// TIA Portal V18 export
FUNCTION_BLOCK "Main_Safety_RTG1"   // FB1, F_LAD
{ S7_Optimized_Access := 'TRUE' }
VERSION : 0.1
// stored: AutoNumber false, IsIECCheckEnabled false, UDAEnableTagReadback false
   VAR
      ACK_GL_Instance : ACK_GL;
      FS_Room1_Instance : "FS_Room1";
      FS_Room2_Instance : "FS_Room2";
      FS_ACC_Instance : "FS_ACC";
      FS_VerticalBeam_Instance : "FS_VerticalBeam";
   END_VAR
BEGIN

REGION Network 1: 全局确认钝化
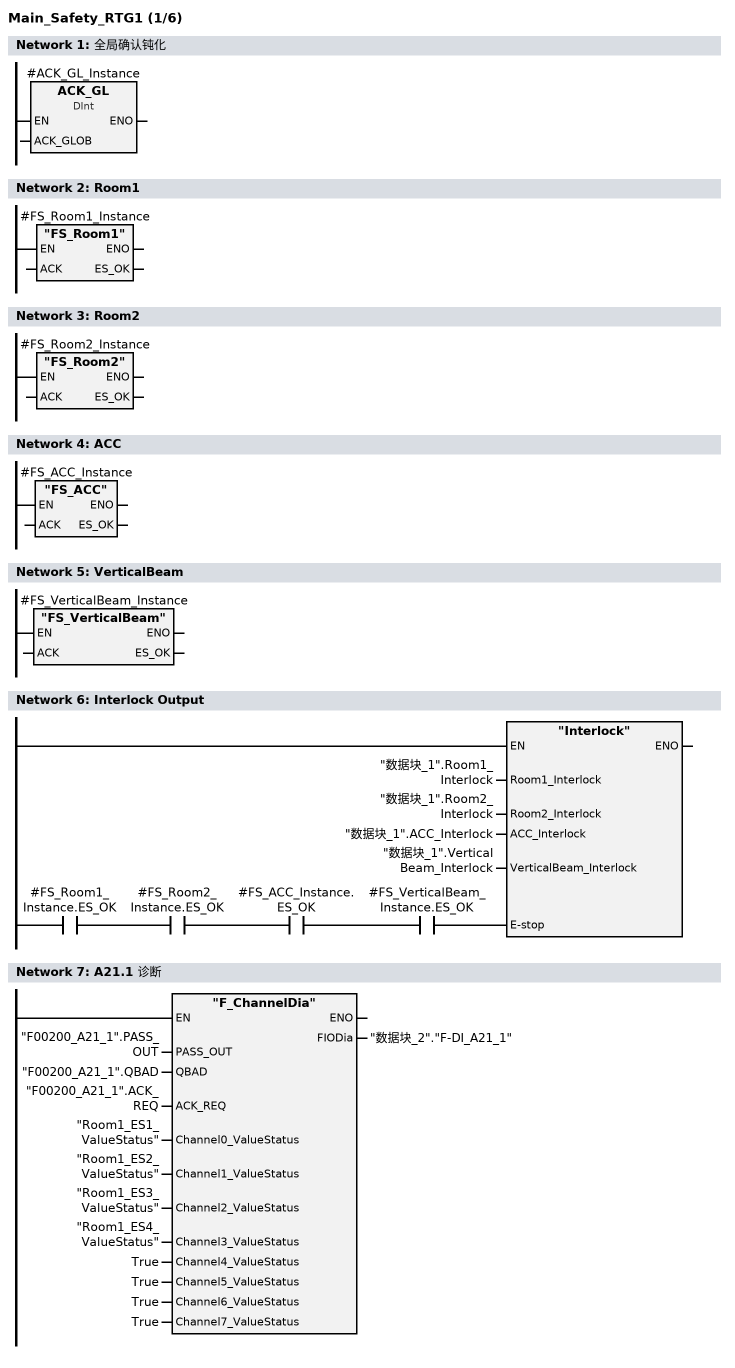
   RUNG wire#powerrail
      { S7_Templates := "codedbool_type := DInt" } #ACK_GL_Instance.ACK_GL(ACK_GLOB :=)
   END_RUNG
   // the same network as SCL:
   #ACK_GL_Instance();   // ACK_GL
END_REGION

REGION Network 2: Room1
   RUNG wire#powerrail
      #FS_Room1_Instance(ACK :=, ES_OK =>)
   END_RUNG
   // the same network as SCL:
   #FS_Room1_Instance();   // "FS_Room1"
END_REGION

REGION Network 3: Room2
   RUNG wire#powerrail
      #FS_Room2_Instance(ACK :=, ES_OK =>)
   END_RUNG
   // the same network as SCL:
   #FS_Room2_Instance();   // "FS_Room2"
END_REGION

REGION Network 4: ACC
   RUNG wire#powerrail
      #FS_ACC_Instance(ACK :=, ES_OK =>)
   END_RUNG
   // the same network as SCL:
   #FS_ACC_Instance();   // "FS_ACC"
END_REGION

REGION Network 5: VerticalBeam
   RUNG wire#powerrail
      #FS_VerticalBeam_Instance(ACK :=, ES_OK =>)
   END_RUNG
   // the same network as SCL:
   #FS_VerticalBeam_Instance();   // "FS_VerticalBeam"
END_REGION

REGION Network 6: Interlock Output
   RUNG wire#powerrail
      "Interlock"(Room1_Interlock := "数据块_1".Room1_Interlock, Room2_Interlock := "数据块_1".Room2_Interlock, ACC_Interlock := "数据块_1".ACC_Interlock, VerticalBeam_Interlock := "数据块_1".VerticalBeam_Interlock, "E-stop" := wire#w1)
   END_RUNG
   RUNG wire#powerrail
      Contact( #FS_Room1_Instance.ES_OK )
      Contact( #FS_Room2_Instance.ES_OK )
      Contact( #FS_ACC_Instance.ES_OK )
      Contact( #FS_VerticalBeam_Instance.ES_OK )
   END_RUNG wire#w1
   // the same network as SCL:
   "Interlock"(Room1_Interlock := "数据块_1".Room1_Interlock,
               Room2_Interlock := "数据块_1".Room2_Interlock,
               ACC_Interlock := "数据块_1".ACC_Interlock,
               VerticalBeam_Interlock := "数据块_1".VerticalBeam_Interlock,
               "E-stop" := #FS_Room1_Instance.ES_OK AND #FS_Room2_Instance.ES_OK AND #FS_ACC_Instance.ES_OK AND #FS_VerticalBeam_Instance.ES_OK);
END_REGION

REGION Network 7: A21.1 诊断
   RUNG wire#powerrail
      "F_ChannelDia"(PASS_OUT := "F00200_A21_1".PASS_OUT, QBAD := "F00200_A21_1".QBAD, ACK_REQ := "F00200_A21_1".ACK_REQ, Channel0_ValueStatus := "Room1_ES1_ValueStatus", Channel1_ValueStatus := "Room1_ES2_ValueStatus", Channel2_ValueStatus := "Room1_ES3_ValueStatus", Channel3_ValueStatus := "Room1_ES4_ValueStatus", Channel4_ValueStatus := True, Channel5_ValueStatus := True, Channel6_ValueStatus := True, Channel7_ValueStatus := True, FIODia => "数据块_2"."F-DI_A21_1")
   END_RUNG
   // the same network as SCL:
   "F_ChannelDia"(PASS_OUT := "F00200_A21_1".PASS_OUT,
                  QBAD := "F00200_A21_1".QBAD,
                  ACK_REQ := "F00200_A21_1".ACK_REQ,
                  Channel0_ValueStatus := "Room1_ES1_ValueStatus",
                  Channel1_ValueStatus := "Room1_ES2_ValueStatus",
                  Channel2_ValueStatus := "Room1_ES3_ValueStatus",
                  Channel3_ValueStatus := "Room1_ES4_ValueStatus",
                  Channel4_ValueStatus := True,
                  Channel5_ValueStatus := True,
                  Channel6_ValueStatus := True,
                  Channel7_ValueStatus := True,
                  FIODia => "数据块_2"."F-DI_A21_1");
END_REGION

REGION Network 8: A21.2 诊断
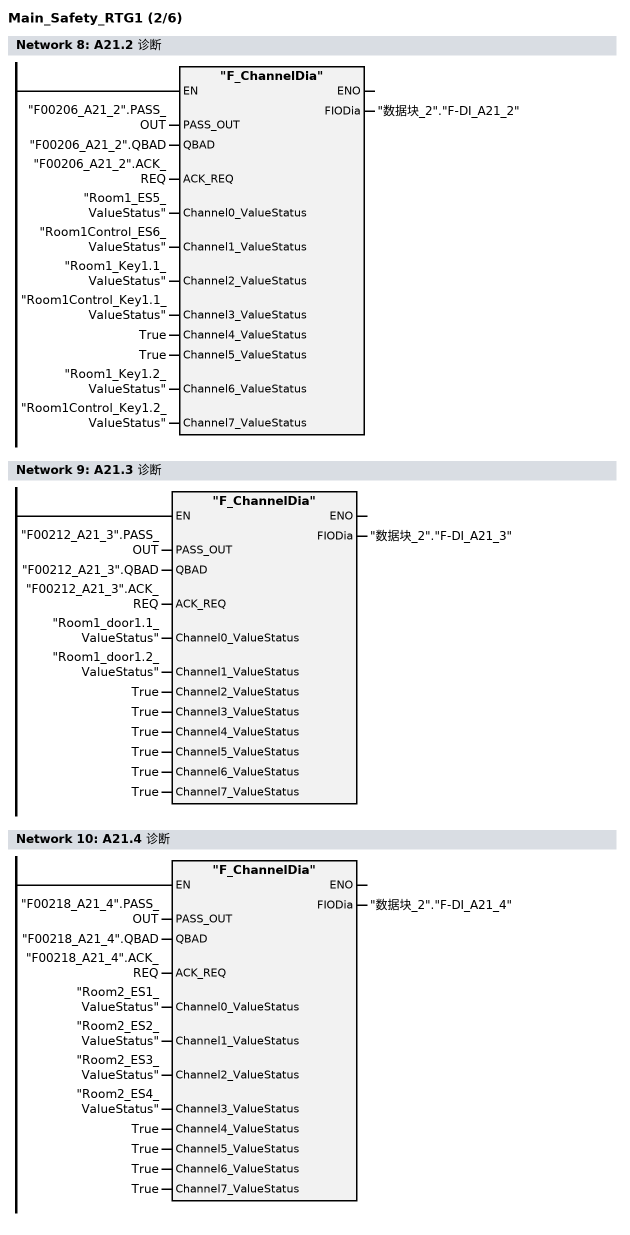
   RUNG wire#powerrail
      "F_ChannelDia"(PASS_OUT := "F00206_A21_2".PASS_OUT, QBAD := "F00206_A21_2".QBAD, ACK_REQ := "F00206_A21_2".ACK_REQ, Channel0_ValueStatus := "Room1_ES5_ValueStatus", Channel1_ValueStatus := "Room1Control_ES6_ValueStatus", Channel2_ValueStatus := "Room1_Key1.1_ValueStatus", Channel3_ValueStatus := "Room1Control_Key1.1_ValueStatus", Channel4_ValueStatus := True, Channel5_ValueStatus := True, Channel6_ValueStatus := "Room1_Key1.2_ValueStatus", Channel7_ValueStatus := "Room1Control_Key1.2_ValueStatus", FIODia => "数据块_2"."F-DI_A21_2")
   END_RUNG
   // the same network as SCL:
   "F_ChannelDia"(PASS_OUT := "F00206_A21_2".PASS_OUT,
                  QBAD := "F00206_A21_2".QBAD,
                  ACK_REQ := "F00206_A21_2".ACK_REQ,
                  Channel0_ValueStatus := "Room1_ES5_ValueStatus",
                  Channel1_ValueStatus := "Room1Control_ES6_ValueStatus",
                  Channel2_ValueStatus := "Room1_Key1.1_ValueStatus",
                  Channel3_ValueStatus := "Room1Control_Key1.1_ValueStatus",
                  Channel4_ValueStatus := True,
                  Channel5_ValueStatus := True,
                  Channel6_ValueStatus := "Room1_Key1.2_ValueStatus",
                  Channel7_ValueStatus := "Room1Control_Key1.2_ValueStatus",
                  FIODia => "数据块_2"."F-DI_A21_2");
END_REGION

REGION Network 9: A21.3 诊断
   RUNG wire#powerrail
      "F_ChannelDia"(PASS_OUT := "F00212_A21_3".PASS_OUT, QBAD := "F00212_A21_3".QBAD, ACK_REQ := "F00212_A21_3".ACK_REQ, Channel0_ValueStatus := "Room1_door1.1_ValueStatus", Channel1_ValueStatus := "Room1_door1.2_ValueStatus", Channel2_ValueStatus := True, Channel3_ValueStatus := True, Channel4_ValueStatus := True, Channel5_ValueStatus := True, Channel6_ValueStatus := True, Channel7_ValueStatus := True, FIODia => "数据块_2"."F-DI_A21_3")
   END_RUNG
   // the same network as SCL:
   "F_ChannelDia"(PASS_OUT := "F00212_A21_3".PASS_OUT,
                  QBAD := "F00212_A21_3".QBAD,
                  ACK_REQ := "F00212_A21_3".ACK_REQ,
                  Channel0_ValueStatus := "Room1_door1.1_ValueStatus",
                  Channel1_ValueStatus := "Room1_door1.2_ValueStatus",
                  Channel2_ValueStatus := True,
                  Channel3_ValueStatus := True,
                  Channel4_ValueStatus := True,
                  Channel5_ValueStatus := True,
                  Channel6_ValueStatus := True,
                  Channel7_ValueStatus := True,
                  FIODia => "数据块_2"."F-DI_A21_3");
END_REGION

REGION Network 10: A21.4 诊断
   RUNG wire#powerrail
      "F_ChannelDia"(PASS_OUT := "F00218_A21_4".PASS_OUT, QBAD := "F00218_A21_4".QBAD, ACK_REQ := "F00218_A21_4".ACK_REQ, Channel0_ValueStatus := "Room2_ES1_ValueStatus", Channel1_ValueStatus := "Room2_ES2_ValueStatus", Channel2_ValueStatus := "Room2_ES3_ValueStatus", Channel3_ValueStatus := "Room2_ES4_ValueStatus", Channel4_ValueStatus := True, Channel5_ValueStatus := True, Channel6_ValueStatus := True, Channel7_ValueStatus := True, FIODia => "数据块_2"."F-DI_A21_4")
   END_RUNG
   // the same network as SCL:
   "F_ChannelDia"(PASS_OUT := "F00218_A21_4".PASS_OUT,
                  QBAD := "F00218_A21_4".QBAD,
                  ACK_REQ := "F00218_A21_4".ACK_REQ,
                  Channel0_ValueStatus := "Room2_ES1_ValueStatus",
                  Channel1_ValueStatus := "Room2_ES2_ValueStatus",
                  Channel2_ValueStatus := "Room2_ES3_ValueStatus",
                  Channel3_ValueStatus := "Room2_ES4_ValueStatus",
                  Channel4_ValueStatus := True,
                  Channel5_ValueStatus := True,
                  Channel6_ValueStatus := True,
                  Channel7_ValueStatus := True,
                  FIODia => "数据块_2"."F-DI_A21_4");
END_REGION

REGION Network 11: A21.5 诊断
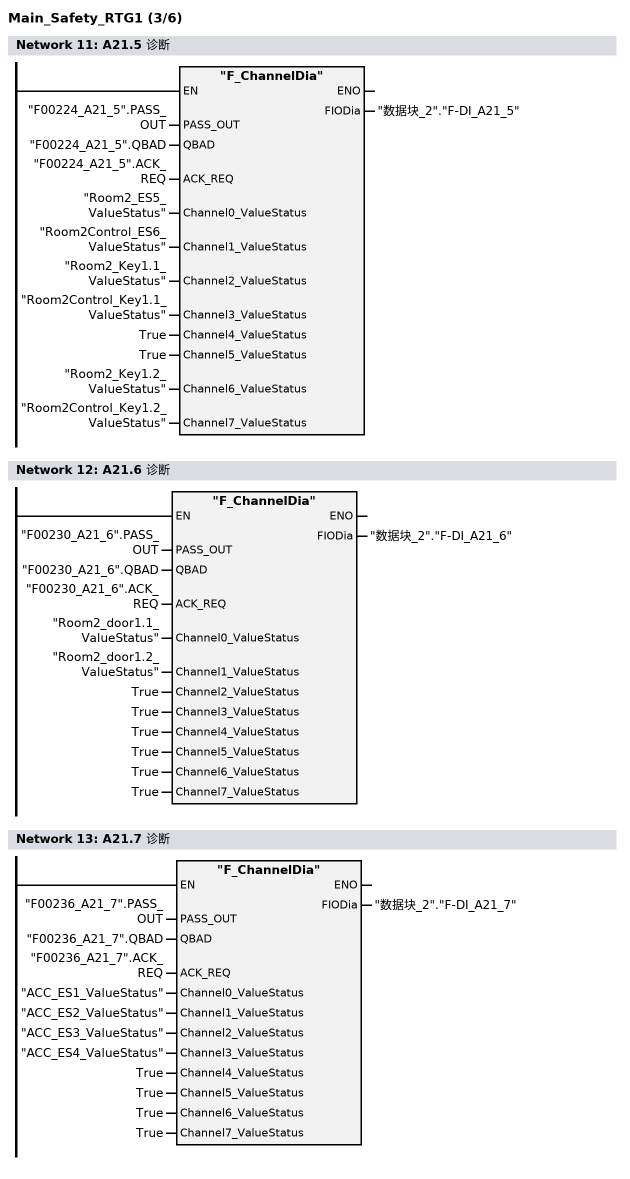
   RUNG wire#powerrail
      "F_ChannelDia"(PASS_OUT := "F00224_A21_5".PASS_OUT, QBAD := "F00224_A21_5".QBAD, ACK_REQ := "F00224_A21_5".ACK_REQ, Channel0_ValueStatus := "Room2_ES5_ValueStatus", Channel1_ValueStatus := "Room2Control_ES6_ValueStatus", Channel2_ValueStatus := "Room2_Key1.1_ValueStatus", Channel3_ValueStatus := "Room2Control_Key1.1_ValueStatus", Channel4_ValueStatus := True, Channel5_ValueStatus := True, Channel6_ValueStatus := "Room2_Key1.2_ValueStatus", Channel7_ValueStatus := "Room2Control_Key1.2_ValueStatus", FIODia => "数据块_2"."F-DI_A21_5")
   END_RUNG
   // the same network as SCL:
   "F_ChannelDia"(PASS_OUT := "F00224_A21_5".PASS_OUT,
                  QBAD := "F00224_A21_5".QBAD,
                  ACK_REQ := "F00224_A21_5".ACK_REQ,
                  Channel0_ValueStatus := "Room2_ES5_ValueStatus",
                  Channel1_ValueStatus := "Room2Control_ES6_ValueStatus",
                  Channel2_ValueStatus := "Room2_Key1.1_ValueStatus",
                  Channel3_ValueStatus := "Room2Control_Key1.1_ValueStatus",
                  Channel4_ValueStatus := True,
                  Channel5_ValueStatus := True,
                  Channel6_ValueStatus := "Room2_Key1.2_ValueStatus",
                  Channel7_ValueStatus := "Room2Control_Key1.2_ValueStatus",
                  FIODia => "数据块_2"."F-DI_A21_5");
END_REGION

REGION Network 12: A21.6 诊断
   RUNG wire#powerrail
      "F_ChannelDia"(PASS_OUT := "F00230_A21_6".PASS_OUT, QBAD := "F00230_A21_6".QBAD, ACK_REQ := "F00230_A21_6".ACK_REQ, Channel0_ValueStatus := "Room2_door1.1_ValueStatus", Channel1_ValueStatus := "Room2_door1.2_ValueStatus", Channel2_ValueStatus := True, Channel3_ValueStatus := True, Channel4_ValueStatus := True, Channel5_ValueStatus := True, Channel6_ValueStatus := True, Channel7_ValueStatus := True, FIODia => "数据块_2"."F-DI_A21_6")
   END_RUNG
   // the same network as SCL:
   "F_ChannelDia"(PASS_OUT := "F00230_A21_6".PASS_OUT,
                  QBAD := "F00230_A21_6".QBAD,
                  ACK_REQ := "F00230_A21_6".ACK_REQ,
                  Channel0_ValueStatus := "Room2_door1.1_ValueStatus",
                  Channel1_ValueStatus := "Room2_door1.2_ValueStatus",
                  Channel2_ValueStatus := True,
                  Channel3_ValueStatus := True,
                  Channel4_ValueStatus := True,
                  Channel5_ValueStatus := True,
                  Channel6_ValueStatus := True,
                  Channel7_ValueStatus := True,
                  FIODia => "数据块_2"."F-DI_A21_6");
END_REGION

REGION Network 13: A21.7 诊断
   RUNG wire#powerrail
      "F_ChannelDia"(PASS_OUT := "F00236_A21_7".PASS_OUT, QBAD := "F00236_A21_7".QBAD, ACK_REQ := "F00236_A21_7".ACK_REQ, Channel0_ValueStatus := "ACC_ES1_ValueStatus", Channel1_ValueStatus := "ACC_ES2_ValueStatus", Channel2_ValueStatus := "ACC_ES3_ValueStatus", Channel3_ValueStatus := "ACC_ES4_ValueStatus", Channel4_ValueStatus := True, Channel5_ValueStatus := True, Channel6_ValueStatus := True, Channel7_ValueStatus := True, FIODia => "数据块_2"."F-DI_A21_7")
   END_RUNG
   // the same network as SCL:
   "F_ChannelDia"(PASS_OUT := "F00236_A21_7".PASS_OUT,
                  QBAD := "F00236_A21_7".QBAD,
                  ACK_REQ := "F00236_A21_7".ACK_REQ,
                  Channel0_ValueStatus := "ACC_ES1_ValueStatus",
                  Channel1_ValueStatus := "ACC_ES2_ValueStatus",
                  Channel2_ValueStatus := "ACC_ES3_ValueStatus",
                  Channel3_ValueStatus := "ACC_ES4_ValueStatus",
                  Channel4_ValueStatus := True,
                  Channel5_ValueStatus := True,
                  Channel6_ValueStatus := True,
                  Channel7_ValueStatus := True,
                  FIODia => "数据块_2"."F-DI_A21_7");
END_REGION

REGION Network 14: A21.8 诊断
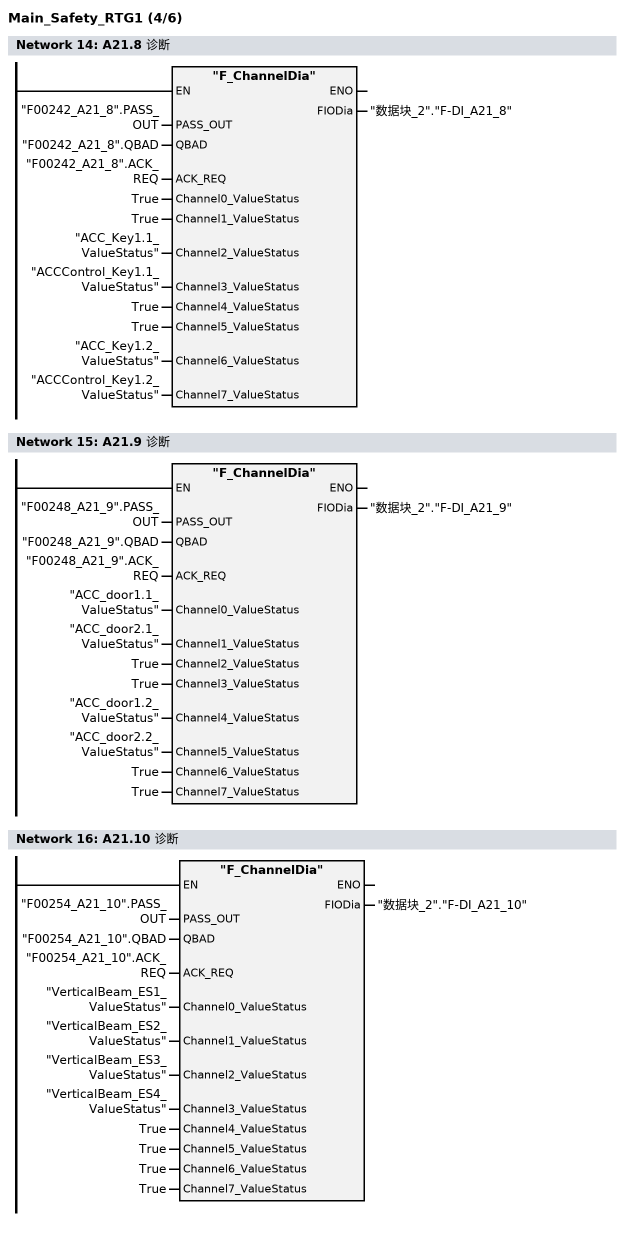
   RUNG wire#powerrail
      "F_ChannelDia"(PASS_OUT := "F00242_A21_8".PASS_OUT, QBAD := "F00242_A21_8".QBAD, ACK_REQ := "F00242_A21_8".ACK_REQ, Channel0_ValueStatus := True, Channel1_ValueStatus := True, Channel2_ValueStatus := "ACC_Key1.1_ValueStatus", Channel3_ValueStatus := "ACCControl_Key1.1_ValueStatus", Channel4_ValueStatus := True, Channel5_ValueStatus := True, Channel6_ValueStatus := "ACC_Key1.2_ValueStatus", Channel7_ValueStatus := "ACCControl_Key1.2_ValueStatus", FIODia => "数据块_2"."F-DI_A21_8")
   END_RUNG
   // the same network as SCL:
   "F_ChannelDia"(PASS_OUT := "F00242_A21_8".PASS_OUT,
                  QBAD := "F00242_A21_8".QBAD,
                  ACK_REQ := "F00242_A21_8".ACK_REQ,
                  Channel0_ValueStatus := True,
                  Channel1_ValueStatus := True,
                  Channel2_ValueStatus := "ACC_Key1.1_ValueStatus",
                  Channel3_ValueStatus := "ACCControl_Key1.1_ValueStatus",
                  Channel4_ValueStatus := True,
                  Channel5_ValueStatus := True,
                  Channel6_ValueStatus := "ACC_Key1.2_ValueStatus",
                  Channel7_ValueStatus := "ACCControl_Key1.2_ValueStatus",
                  FIODia => "数据块_2"."F-DI_A21_8");
END_REGION

REGION Network 15: A21.9 诊断
   RUNG wire#powerrail
      "F_ChannelDia"(PASS_OUT := "F00248_A21_9".PASS_OUT, QBAD := "F00248_A21_9".QBAD, ACK_REQ := "F00248_A21_9".ACK_REQ, Channel0_ValueStatus := "ACC_door1.1_ValueStatus", Channel1_ValueStatus := "ACC_door2.1_ValueStatus", Channel2_ValueStatus := True, Channel3_ValueStatus := True, Channel4_ValueStatus := "ACC_door1.2_ValueStatus", Channel5_ValueStatus := "ACC_door2.2_ValueStatus", Channel6_ValueStatus := True, Channel7_ValueStatus := True, FIODia => "数据块_2"."F-DI_A21_9")
   END_RUNG
   // the same network as SCL:
   "F_ChannelDia"(PASS_OUT := "F00248_A21_9".PASS_OUT,
                  QBAD := "F00248_A21_9".QBAD,
                  ACK_REQ := "F00248_A21_9".ACK_REQ,
                  Channel0_ValueStatus := "ACC_door1.1_ValueStatus",
                  Channel1_ValueStatus := "ACC_door2.1_ValueStatus",
                  Channel2_ValueStatus := True,
                  Channel3_ValueStatus := True,
                  Channel4_ValueStatus := "ACC_door1.2_ValueStatus",
                  Channel5_ValueStatus := "ACC_door2.2_ValueStatus",
                  Channel6_ValueStatus := True,
                  Channel7_ValueStatus := True,
                  FIODia => "数据块_2"."F-DI_A21_9");
END_REGION

REGION Network 16: A21.10 诊断
   RUNG wire#powerrail
      "F_ChannelDia"(PASS_OUT := "F00254_A21_10".PASS_OUT, QBAD := "F00254_A21_10".QBAD, ACK_REQ := "F00254_A21_10".ACK_REQ, Channel0_ValueStatus := "VerticalBeam_ES1_ValueStatus", Channel1_ValueStatus := "VerticalBeam_ES2_ValueStatus", Channel2_ValueStatus := "VerticalBeam_ES3_ValueStatus", Channel3_ValueStatus := "VerticalBeam_ES4_ValueStatus", Channel4_ValueStatus := True, Channel5_ValueStatus := True, Channel6_ValueStatus := True, Channel7_ValueStatus := True, FIODia => "数据块_2"."F-DI_A21_10")
   END_RUNG
   // the same network as SCL:
   "F_ChannelDia"(PASS_OUT := "F00254_A21_10".PASS_OUT,
                  QBAD := "F00254_A21_10".QBAD,
                  ACK_REQ := "F00254_A21_10".ACK_REQ,
                  Channel0_ValueStatus := "VerticalBeam_ES1_ValueStatus",
                  Channel1_ValueStatus := "VerticalBeam_ES2_ValueStatus",
                  Channel2_ValueStatus := "VerticalBeam_ES3_ValueStatus",
                  Channel3_ValueStatus := "VerticalBeam_ES4_ValueStatus",
                  Channel4_ValueStatus := True,
                  Channel5_ValueStatus := True,
                  Channel6_ValueStatus := True,
                  Channel7_ValueStatus := True,
                  FIODia => "数据块_2"."F-DI_A21_10");
END_REGION

REGION Network 17: A21.11 诊断
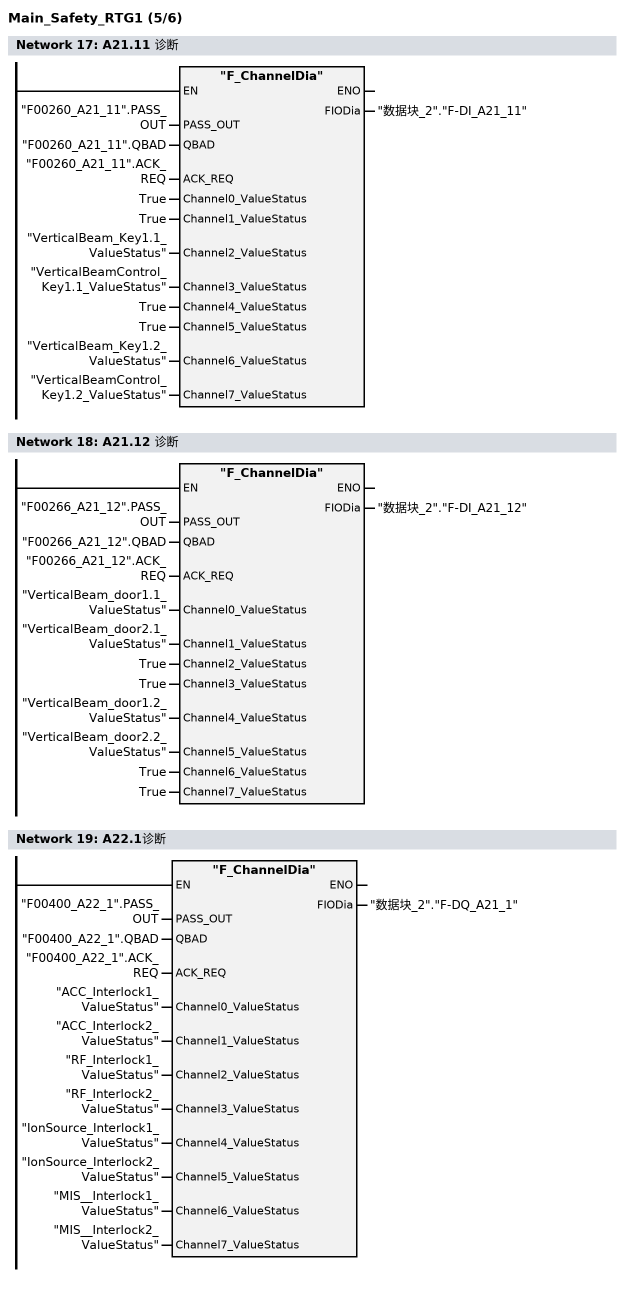
   RUNG wire#powerrail
      "F_ChannelDia"(PASS_OUT := "F00260_A21_11".PASS_OUT, QBAD := "F00260_A21_11".QBAD, ACK_REQ := "F00260_A21_11".ACK_REQ, Channel0_ValueStatus := True, Channel1_ValueStatus := True, Channel2_ValueStatus := "VerticalBeam_Key1.1_ValueStatus", Channel3_ValueStatus := "VerticalBeamControl_Key1.1_ValueStatus", Channel4_ValueStatus := True, Channel5_ValueStatus := True, Channel6_ValueStatus := "VerticalBeam_Key1.2_ValueStatus", Channel7_ValueStatus := "VerticalBeamControl_Key1.2_ValueStatus", FIODia => "数据块_2"."F-DI_A21_11")
   END_RUNG
   // the same network as SCL:
   "F_ChannelDia"(PASS_OUT := "F00260_A21_11".PASS_OUT,
                  QBAD := "F00260_A21_11".QBAD,
                  ACK_REQ := "F00260_A21_11".ACK_REQ,
                  Channel0_ValueStatus := True,
                  Channel1_ValueStatus := True,
                  Channel2_ValueStatus := "VerticalBeam_Key1.1_ValueStatus",
                  Channel3_ValueStatus := "VerticalBeamControl_Key1.1_ValueStatus",
                  Channel4_ValueStatus := True,
                  Channel5_ValueStatus := True,
                  Channel6_ValueStatus := "VerticalBeam_Key1.2_ValueStatus",
                  Channel7_ValueStatus := "VerticalBeamControl_Key1.2_ValueStatus",
                  FIODia => "数据块_2"."F-DI_A21_11");
END_REGION

REGION Network 18: A21.12 诊断
   RUNG wire#powerrail
      "F_ChannelDia"(PASS_OUT := "F00266_A21_12".PASS_OUT, QBAD := "F00266_A21_12".QBAD, ACK_REQ := "F00266_A21_12".ACK_REQ, Channel0_ValueStatus := "VerticalBeam_door1.1_ValueStatus", Channel1_ValueStatus := "VerticalBeam_door2.1_ValueStatus", Channel2_ValueStatus := True, Channel3_ValueStatus := True, Channel4_ValueStatus := "VerticalBeam_door1.2_ValueStatus", Channel5_ValueStatus := "VerticalBeam_door2.2_ValueStatus", Channel6_ValueStatus := True, Channel7_ValueStatus := True, FIODia => "数据块_2"."F-DI_A21_12")
   END_RUNG
   // the same network as SCL:
   "F_ChannelDia"(PASS_OUT := "F00266_A21_12".PASS_OUT,
                  QBAD := "F00266_A21_12".QBAD,
                  ACK_REQ := "F00266_A21_12".ACK_REQ,
                  Channel0_ValueStatus := "VerticalBeam_door1.1_ValueStatus",
                  Channel1_ValueStatus := "VerticalBeam_door2.1_ValueStatus",
                  Channel2_ValueStatus := True,
                  Channel3_ValueStatus := True,
                  Channel4_ValueStatus := "VerticalBeam_door1.2_ValueStatus",
                  Channel5_ValueStatus := "VerticalBeam_door2.2_ValueStatus",
                  Channel6_ValueStatus := True,
                  Channel7_ValueStatus := True,
                  FIODia => "数据块_2"."F-DI_A21_12");
END_REGION

REGION Network 19: A22.1诊断
   RUNG wire#powerrail
      "F_ChannelDia"(PASS_OUT := "F00400_A22_1".PASS_OUT, QBAD := "F00400_A22_1".QBAD, ACK_REQ := "F00400_A22_1".ACK_REQ, Channel0_ValueStatus := "ACC_Interlock1_ValueStatus", Channel1_ValueStatus := "ACC_Interlock2_ValueStatus", Channel2_ValueStatus := "RF_Interlock1_ValueStatus", Channel3_ValueStatus := "RF_Interlock2_ValueStatus", Channel4_ValueStatus := "IonSource_Interlock1_ValueStatus", Channel5_ValueStatus := "IonSource_Interlock2_ValueStatus", Channel6_ValueStatus := "MIS__Interlock1_ValueStatus", Channel7_ValueStatus := "MIS__Interlock2_ValueStatus", FIODia => "数据块_2"."F-DQ_A21_1")
   END_RUNG
   // the same network as SCL:
   "F_ChannelDia"(PASS_OUT := "F00400_A22_1".PASS_OUT,
                  QBAD := "F00400_A22_1".QBAD,
                  ACK_REQ := "F00400_A22_1".ACK_REQ,
                  Channel0_ValueStatus := "ACC_Interlock1_ValueStatus",
                  Channel1_ValueStatus := "ACC_Interlock2_ValueStatus",
                  Channel2_ValueStatus := "RF_Interlock1_ValueStatus",
                  Channel3_ValueStatus := "RF_Interlock2_ValueStatus",
                  Channel4_ValueStatus := "IonSource_Interlock1_ValueStatus",
                  Channel5_ValueStatus := "IonSource_Interlock2_ValueStatus",
                  Channel6_ValueStatus := "MIS__Interlock1_ValueStatus",
                  Channel7_ValueStatus := "MIS__Interlock2_ValueStatus",
                  FIODia => "数据块_2"."F-DQ_A21_1");
END_REGION

REGION Network 20: A22.2诊断
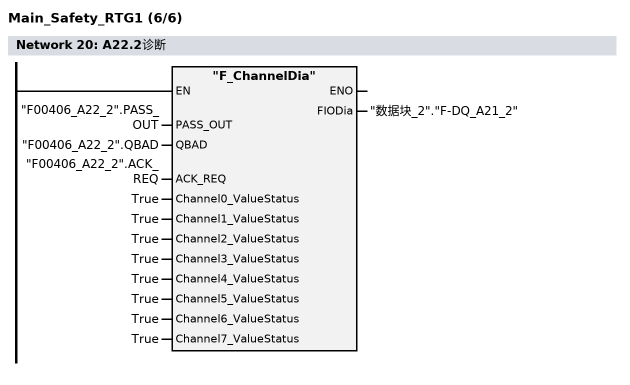
   RUNG wire#powerrail
      "F_ChannelDia"(PASS_OUT := "F00406_A22_2".PASS_OUT, QBAD := "F00406_A22_2".QBAD, ACK_REQ := "F00406_A22_2".ACK_REQ, Channel0_ValueStatus := True, Channel1_ValueStatus := True, Channel2_ValueStatus := True, Channel3_ValueStatus := True, Channel4_ValueStatus := True, Channel5_ValueStatus := True, Channel6_ValueStatus := True, Channel7_ValueStatus := True, FIODia => "数据块_2"."F-DQ_A21_2")
   END_RUNG
   // the same network as SCL:
   "F_ChannelDia"(PASS_OUT := "F00406_A22_2".PASS_OUT,
                  QBAD := "F00406_A22_2".QBAD,
                  ACK_REQ := "F00406_A22_2".ACK_REQ,
                  Channel0_ValueStatus := True,
                  Channel1_ValueStatus := True,
                  Channel2_ValueStatus := True,
                  Channel3_ValueStatus := True,
                  Channel4_ValueStatus := True,
                  Channel5_ValueStatus := True,
                  Channel6_ValueStatus := True,
                  Channel7_ValueStatus := True,
                  FIODia => "数据块_2"."F-DQ_A21_2");
END_REGION
END_FUNCTION_BLOCK
